KUKA KRL program: delmens.src

&ACCESS RVO3
&REL 2
&PARAM TEMPLATE = C:\KRC\Roboter\Template\vorgabe
&PARAM EDITMASK = *
DEF DelMens( )

$MSG_T.RELEASE=TRUE
WHILE $MSG_T.VALID==TRUE
;FOLD WAIT Time= 0.5 sec;%{PE}%R 4.1.16,%MKUKATPBASIS,%CWAIT,%VWAIT,%P 2:0.5
WAIT SEC 0.5
;ENDFOLD
$MSG_T.VALID=FALSE
ENDWHILE

END
